Omron CX-Programmer project NewProject (CX-Programmer 9.75)

# PLC LED_PROJECT: CJ2M CPU11

## Global symbols (name address type ; comment)
0.00 BOOL  ; START/STOP
0.01 BOOL  ; INC BUTTON
0.02 BOOL  ; DEC BUTTON
100.00 BOOL  ; LED
T0000 BOOL  ; T0

## Program NewProgram1 (cyclic task 0)
Local symbols
K10 INT
k10 UINT_BCD

### Section Section1

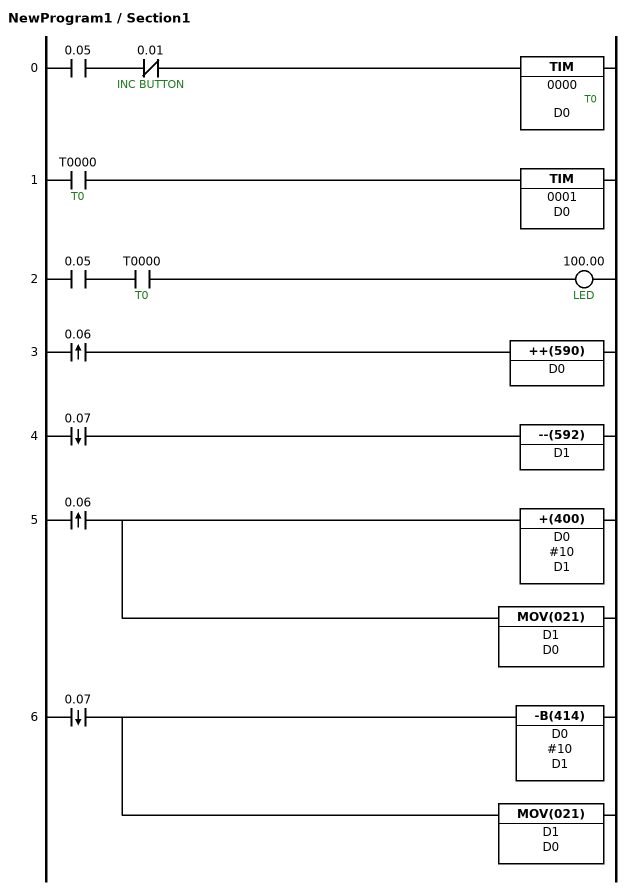
; rung 0
LD 0.05
ANDNOT 0.01  ; INC BUTTON
TIM 0000 D0  ; T0
; rung 1
LD T0000  ; T0
TIM 0001 D0
; rung 2
LD 0.05
AND T0000  ; T0
OUT 100.00  ; LED
; rung 3
@LD 0.06
++(590) D0
; rung 4
%LD 0.07
--(592) D1
; rung 5
@LD 0.06
+(400) D0 #10 D1
MOV(021) D1 D0
; rung 6
%LD 0.07
-B(414) D0 #10 D1
MOV(021) D1 D0

### Section END
; rung 0
END(001)